INTERFACE I_Input

METHOD Pause : I_Output
VAR_INPUT
	bPause 		:  BOOL; // Pause Timer (TRUE), Only Pauses if IN := TRUE.
END_VAR
END_METHOD

METHOD Start : I_Output
VAR_INPUT
	bStart 		: BOOL;  // Starts timer with rising edge, resets timer with falling edge.
END_VAR
END_METHOD

METHOD StartTimer : I_Output
VAR_INPUT
END_VAR
END_METHOD

METHOD StopTimer : I_Output
VAR_INPUT
END_VAR
END_METHOD

END_INTERFACE

(* stored: Version 1.1.0.1, ProductVersion 3.1.4024.12
   Itf I_Input: Id {1df94bf4-5590-48f5-97b2-bce8c32c17ba}
   Method Pause: Id {bb623033-c04f-44ec-b93a-dec8f1de4c22}
   Method Start: Id {85832a66-a4f9-4ebb-a085-bf5e6ddc16eb}
   Method StartTimer: Id {a05f3310-647c-48ea-812b-1aa4bfff9e2e}
   Method StopTimer: Id {36bdef81-9090-4b12-b1e3-0d93056e4904} *)
